FUNCTION_BLOCK Q_NumericValue_PHYSA (* Command change numeric value — accepts physical REAL value via AR adapter (wraps Q_NumericValue_PHYS) *)
  (* Standard: ISO 11783-6; Description: Copyright (c) 2026 Meisterschulen am Ostbahnhof This program and the accompanying materials are made available under the terms of the Eclipse Public License 2.0 which is available at https://www.eclipse.org/legal/epl-2.0/ SPDX-License-Identifier: EPL-2.0 *)
  (* Version 1.0, 2026-04-14, Franz Höpfinger, Meisterschulen am Ostbahnhof, initial API and implementation and/or initial documentation *)
  PACKAGE isobus::UT::Q;
  IMPORT isobus::UT::Q::const::IDs::ID_NULL;
  IMPORT logiBUS::utils::conversion::phys::NumericObjectPool_S;
  (* Documentation:
  Command change numeric value ( Part 6 - F.22 ) — physical-value AR adapter wrapper
   This FB is an AR adapter wrapper around Q_NumericValue_PHYS (which in turn wraps Q_NumericValue). The physical REAL value is supplied via the rPhys AR adapter socket, the object pool properties (including stObj.u16ObjId) via INIT. Limit violations are reported on the xOver/xUnder AX adapter plugs.
   Valid Object IDs
   stObj.u16ObjId is valid if it falls within one of the following ISO 11783-6 ID ranges (Annex F.22 — see Q_NumericValue):
    - InputBooleanField: 7000 – 7999
   - InputNumberField: 9000 – 9999
   - InputListField: 10000 – 10999
   - OutputNumberField: 12000 – 12999
   - Meter: 17000 – 17999
   - LinearBarGraph: 18000 – 18999
   - ArchedBarGraph: 19000 – 19999
   - NumberVariable: 21000 – 21999
   - ObjectPointer: 27000 – 27999
   - OutputListObject: 37000 – 37999
   - ExternalObjectPointer: 43000 – 43999
   - AnimationObject: 44000 – 44999
   - ScaledGraphicObject: 48000 – 48999
    ID_NULL (65535) is not a command target but can be used in stObj.u16ObjId via INIT to deactivate the FB. Any ID outside these ranges is invalid for commanding. The result codes (s16result) are identical to Q_NumericValue.
  *)
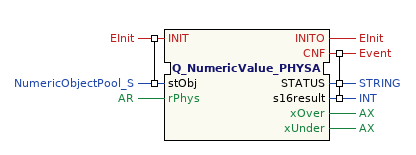
  EVENT_INPUT
    INIT : EInit WITH stObj; (* Service Initialization *)
  END_EVENT
  EVENT_OUTPUT
    INITO : EInit; (* Initialization Confirm *)
    CNF WITH STATUS, s16result; (* Confirmation of Requested Service *)
  END_EVENT
  VAR_INPUT
    stObj : logiBUS::utils::conversion::phys::NumericObjectPool_S := (u16ObjId := ID_NULL, r32Scale := 1.0, i32Offset := 0, u8Decimals := 0); (* Object pool properties (u16ObjId, scale, offset, decimals) *)
  END_VAR
  VAR_OUTPUT
    STATUS : STRING; (* Service Status *)
    s16result : INT; (* retval see Q_NumericValue *)
  END_VAR
  SOCKETS
    rPhys : adapter::types::unidirectional::AR; (* Physical REAL value input *)
  END_SOCKETS
  PLUGS
    xOver : adapter::types::unidirectional::AX; (* Physical value exceeds upper ISOBUS limit *)
    xUnder : adapter::types::unidirectional::AX; (* Physical value below lower ISOBUS limit *)
  END_PLUGS
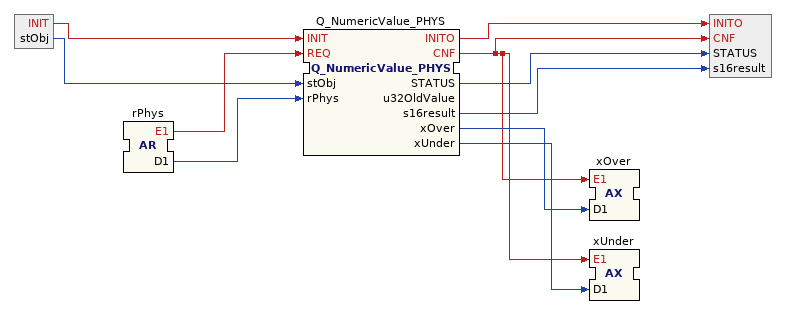
  FBS
    Q_NumericValue_PHYS : isobus::UT::Q::Q_NumericValue_PHYS;
  END_FBS
  EVENT_CONNECTIONS
    INIT TO Q_NumericValue_PHYS.INIT;
    rPhys.E1 TO Q_NumericValue_PHYS.REQ;
    Q_NumericValue_PHYS.INITO TO INITO;
    Q_NumericValue_PHYS.CNF TO CNF;
    Q_NumericValue_PHYS.CNF TO xOver.E1;
    Q_NumericValue_PHYS.CNF TO xUnder.E1;
  END_CONNECTIONS
  DATA_CONNECTIONS
    stObj TO Q_NumericValue_PHYS.stObj;
    rPhys.D1 TO Q_NumericValue_PHYS.rPhys;
    Q_NumericValue_PHYS.STATUS TO STATUS;
    Q_NumericValue_PHYS.s16result TO s16result;
    Q_NumericValue_PHYS.xOver TO xOver.D1;
    Q_NumericValue_PHYS.xUnder TO xUnder.D1;
  END_CONNECTIONS
END_FUNCTION_BLOCK
